// TIA Portal V19 export
TYPE "RTrk_Item"
   STRUCT
      ID_R : DInt;   // ID della coppia di fori di riferimento
      PNo : DInt;
      WL_Indx : DInt;
      WL_Part : DInt;
      BeginPos : LReal;   // Poisione inizio pezzo su materiale in profilatrice
      EndPos : LReal;   // Posizione fine parte
      Quality : Int;
   END_STRUCT;
END_TYPE
